// Mitsubishi GX Works2 project: math01   PLC: Q02/Q02H

PROGRAM MAIN
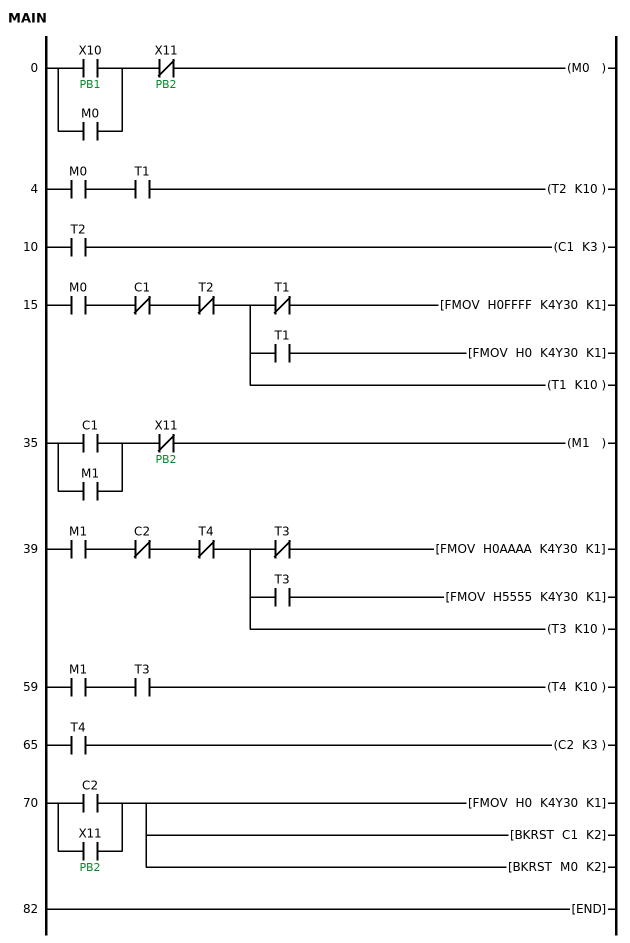
0     LD      X10  ; PB1
      OR      M0
      ANI     X11  ; PB2
      OUT     M0
4     LD      M0
      AND     T1
      OUT     T2 K10
10    LD      T2
      OUT     C1 K3
15    LD      M0
      ANI     C1
      ANI     T2
      MPS
      ANI     T1
      FMOV    H0FFFF K4Y30 K1
      MRD
      AND     T1
      FMOV    H0 K4Y30 K1
      MPP
      OUT     T1 K10
35    LD      C1
      OR      M1
      ANI     X11  ; PB2
      OUT     M1
39    LD      M1
      ANI     C2
      ANI     T4
      MPS
      ANI     T3
      FMOV    H0AAAA K4Y30 K1
      MRD
      AND     T3
      FMOV    H5555 K4Y30 K1
      MPP
      OUT     T3 K10
59    LD      M1
      AND     T3
      OUT     T4 K10
65    LD      T4
      OUT     C2 K3
70    LD      C2
      OR      X11  ; PB2
      FMOV    H0 K4Y30 K1
      BKRST   C1 K2
      BKRST   M0 K2
82    END
END_PROGRAM

// device comments not shown above
X0  ; 공급_후
X1  ; 공급_전
X2  ; 드릴_상
X3  ; 드릴_하
X4  ; 송출_후
X5  ; 송출_전
X6  ; 배출_후
X7  ; 배출_전
X8  ; 매거진
X9  ; 비금속
X0A  ; 금속
X12  ; PB3
Y20  ; 공급_전
Y21  ; 공급_후
Y22  ; 드릴_하강
Y23  ; 송출_전
Y24  ; 송출_후
Y25  ; 배출_전
Y26  ; 배출_후
Y27  ; 컨베어
Y28  ; 가공드
Y29  ; 적색
Y2A  ; 황색
Y2B  ; 녹색
